TYPE FactoryIO_Output :
STRUCT
	bStopBlade		:	BOOL;
	bStartLight		:	BOOL;
	bResetLight		:	BOOL;
	bStopLight		:	BOOL;
	nBufferConveyor	: 	WORD;
	nExitConveyor	: 	WORD;
	nCounter		:	WORD;
END_STRUCT
END_TYPE

(* stored: Version 1.1.0.1, ProductVersion 3.1.4024.12
   DUT FactoryIO_Output: Id {62515850-4fb1-4aa1-b1cd-dee53f154e17} *)
